TYPE ST_GateValve :
STRUCT
	biSnGateValve_Close:BOOL;
	biSnGateValve_Open:BOOL;
	boCylGateValve_Close:BOOL;
	boCylGateValve_Open:BOOL;
END_STRUCT
END_TYPE

(* stored: Version 1.1.0.1, ProductVersion 3.1.4024.12
   DUT ST_GateValve: Id {62dfd8e4-3bd9-44a4-8fb2-5421e3124c21} *)
